FUNCTION FN_NumToLane : cLaneSel
VAR_INPUT
	Lane: DINT;
END_VAR

//Determin lane from string input
IF Lane = cLaneSel.Green THEN
	FN_NumToLane := cLaneSel.Green;
ELSIF Lane = cLaneSel.Red THEN
	FN_NumToLane := cLaneSel.Red;
ELSIF Lane = cLaneSel.Blue THEN
	FN_NumToLane := cLaneSel.Blue;
ELSE
	FN_NumToLane := cLaneSel.None;
END_IF

END_FUNCTION

(* stored: Version 1.1.0.1, ProductVersion 3.1.4024.6
   POU FN_NumToLane: Id {c426b26a-7054-49fa-a538-65091a9d2dd0}, SpecialFunc None *)
